Staubli VAL3: RobotPolish.pjx

--- RobotPolish.pjx ---
Parameters version=s7.3 stackSize=5000 millimeterUnit=true
Program file=DeleteTxt.pgx
Program file=Kill.pgx
Program file=Poll.pgx
Program file=_refreshDebugPa.pgx
Program file=alarm_action.pgx
Program file=checkIn.pgx
Program file=checkOut.pgx
Program file=check_PC.pgx
Program file=goHome.pgx
Program file=init.pgx
Program file=logandpopMsg.pgx
Program file=main.pgx
Program file=massage.pgx
Program file=page_debug.pgx
Program file=page_main.pgx
Program file=page_production.pgx
Program file=page_setHome.pgx
Program file=page_setSpdVal.pgx
Program file=page_txtSelect.pgx
Program file=prdMassage.pgx
Program file=prdStatusList.pgx
Program file=prd_action.pgx
Program file=production.pgx
Program file=readForce.pgx
Program file=resumeProduct.pgx
Program file=start.pgx
Program file=stop.pgx
Program file=userInterface.pgx
Data file=RobotPolish.dtx
Library alias=read path=Disk://readText/readText.pjx autoload=true password=
Library alias=io path=Disk://IO/IO.pjx autoload=true password=
Library alias=ati path=Disk://atiForceSen7/atiForceSen7.pjx autoload=true password=
Library alias=use path=Disk://userPage/userPage.pjx autoload=true password=
Library alias=date path=Disk://dateBase/dateBase.pjx autoload=true password=
Library alias=setFrm path=Disk://CircleCenter/CircleCenter.pjx autoload=true password=
Library alias=UI path=Disk://StaubliUI/StaubliUI.pjx autoload=true password=
Library alias=CalTool path=Disk://StaubliCalTool7/StaubliCalTool7.pjx autoload=true password=

--- RobotPolish.dtx ---
bool bBIO[32]
  [16] = true
  [18] = true
  [22] = true
bool bDebug_PC[6] = true
bool bExit = true
bool bForceError
bool bHome
bool bInterVal
bool bIsAlarm
bool bIsPower = true
bool bJntOrPtSpd
bool bOverRun
bool bPause
bool bRefreshMsg[6]
  [0] = true
  [1] = true
  [2] = true
  [3] = true
  [4] = true
  [5] = true
bool bSuspend = true
bool bTableAlm
bool bTxtLoad
bool bUpload
bool bZero
frame fFrame = {x=1612.970915, y=39.891118, z=-82.912831, rx=0.071185, ry=-0.543234, rz=-77.228709, fatherId=world[0]}
jointRx jCurrentJoint = {j1=8.22, j2=20.1, j3=107.19, j4=-141.77, j5=44.38, j6=150.9}
jointRx jHome = {j1=40.634813, j2=24.616005, j3=104.715218, j4=-108.663007, j5=68.526435, j6=132.709111}
jointRx jJHome = {j1=11.40774, j2=30.671658, j3=109.333141, j4=204.624689, j5=51.130912, j6=-196.428273}
mdesc mNomSpeed = {accel=36, vel=60, decel=36, rmax=2000, tmax=100, blend=cartesian, leave=5, reach=5}
num nATIPress
num nATiPressBuff
num nFunctionIndex = -1
num nInterfaceType = 9
num nJntList
public num nLimitAti[6]
  [0] = 500
  [1] = 500
  [2] = 500
  [3] = 100
  [4] = 100
  [5] = 100
num nMoveID
num nPage
num nPauseTime = 6
num nSelect
num nTabSpeed = 5
num nTimeBuff = 6728.108
num nTxtSelseted = 3
num nVirtualKey = -1
num nWorkModeStatus
num nWorkingMode = 4
pointRx p = {x=-96.25, y=181, rx=-8.631, ry=175.438, rz=-89.108, fatherId=fFrame[0]}
pointRx pCurrent = {x=-7.439422, y=-0.703489, z=141.92314, rx=-0.008216, ry=-179.493493, rz=-59.800957, shoulder=lefty, elbow=epositive, wrist=wpositive, fatherId=fFrame[0]}
string sButtons[2]
  [0] = "Yes"
  [1] = "No"
string sErrorMsg[8]
  [0] = "UPS报错，检查工厂供电"
  [1] = "转台故障报警"
  [2] = "工具报警"
  [3] = "ATI与机器人通讯异常"
  [4] = "打磨力超出上限"
  [5] = "急停状态激活中"
string sItems[8]
  [0] = "信号"
  [1] = "生产"
  [2] = "TCP"
  [3] = "Frame"
  [4] = "Home"
  [5] = "速度"
  [7] = "退出"
string sMassage
string sPrdStatus[10]
  [0] = "Txt文件:"
  [1] = "TEST.txt"
  [2] = "生产状态:无生产"
  [3] = "运动状态:Move"
  [4] = "总路径个数:     1"
  [5] = "当前路径  :     1"
  [6] = "写入点个数:   902"
  [7] = "读取点个数:     1"
  [8] = "当前MoveID:     0"
  [9] = "瞬时速度  :  5.4 "
string sStrFileName[6]
  [0] = "1233"
  [1] = "BUFF"
  [2] = "TEST.txt"
  [3] = "speed of TCP.txt"
string sTxtLists[12]
  [0] = "1233"
  [1] = "BUFF"
  [2] = "TEST"
  [3] = "TEST.txt"
  [4] = "speed of TCP.txt"
string sTxtSelected = "TEST.txt"
tool tTTool = {x=1.417, y=48.029, z=261.326, rx=-28.407, ry=-42.029, rz=-19.448, fatherId=flange[0], ioLink=valve1}
public tool tTool = {x=350.22, y=-0.767094, z=232.538993, rx=-89.841339, ry=89.729222, rz=89.842087, fatherId=flange[0], ioLink=valve1}
trsf trFrame = {x=1460.596362, y=35.712914, z=-199.189903, rx=-0.117127, ry=-0.30554, rz=-53.750077}

--- main.pgx ---
program main()
begin

  //初始化
  call DeleteTxt()
  call init()
  //创建同步任务,机器人实时读取ATI传感器数据
  //2015.06.23
  //taskCreateSync "readAtiForce",0.05,bOverRun,readForce()
  taskCreate "readAtiForce",100,readForce()


  //创建任务,实时扫描输入输出信号
  //当date:bPLC变量为true时,调用真实机器人联机调试程序;
  //当date:bPLC变量为false时,调用PC模拟程序;
  if date:bPLC
    taskCreate "Input",96,checkIn()
    taskCreate "Output",98,checkOut()
  else
    taskCreate "PC_IO",98,check_PC()
  endIf
  //创建任务,用户操作界面
  taskCreate "HMI",85,userInterface()



end

--- check_PC.pgx ---
program check_PC()
  local jointRx l_jCurrent
  local bool l_bRefresh
begin
  while !bExit

    //工厂断电报警
    if bDebug_PC[0]==false
      call logandpopMsg(sErrorMsg[0],bRefreshMsg[0])
      if read:bCycle
        call alarm_action()
      endIf
      if workingMode()==4
        disablePower()
      endIf
    else
      bRefreshMsg[0]=true
    endIf

    //check
    call Poll()
    //

    //转台故障信号
    //    if dioGet(io:doB_9_tableOn)==1
    //      if dioGet(io:doB_0_speed)==1 or dioGet(io:doB_1_speed)==1 or dioGet(io:doB_2_speed)==1 or dioGet(io:doB_3_speed)==1 or dioGet(io:doB_4_speed)==1 or dioGet(io:doB_5_speed)==1
    //        bTableAlm=!watch(dioGet(io:diB_2_tableOn)==1,2)
    //        if !bTableAlm
    //          bRefreshMsg[1]=true
    //        else
    //          call logandpopMsg(sErrorMsg[1],bRefreshMsg[1])
    //          if read:bCycle
    //            call alarm_action()
    //          endIf
    //        endIf
    //      else
    //        bTableAlm=false
    //      endIf
    //    else
    //      bTableAlm=false
    //    endIf
    //工具报警信号
    if bDebug_PC[2]==true
      call logandpopMsg(sErrorMsg[2],bRefreshMsg[2])
      if read:bCycle
        call alarm_action()
      endIf
    else
      bRefreshMsg[2]=true
    endIf
    //ATI通讯状态检测
    if bDebug_PC[3]==true
      call logandpopMsg(sErrorMsg[3],bRefreshMsg[3])
      if read:bCycle
        call alarm_action()
      endIf
    else
      bRefreshMsg[3]=true
    endIf
    //传感器力/扭矩上限检测
    //需要根据测试结果设置力及力矩上限
    if bDebug_PC[4]==true
      bForceError=true
      call logandpopMsg(sErrorMsg[4],bRefreshMsg[4])
      if read:bCycle
        call alarm_action()
      endIf
    else
      bForceError=false
      bRefreshMsg[4]=true
    endIf
    //急停处理
    if esStatus()==2
      call logandpopMsg(sErrorMsg[5],bRefreshMsg[5])
      call prd_action("急停处理")
    else
      bRefreshMsg[5]=true
    endIf
    //远程上电
    if workingMode(nWorkModeStatus)==4 and dioGet(io:diB_0_UPS)==0
      if dioGet(io:doB_10_systeAlm)==0
        enablePower()
        dioSet(io:doB_6_toolPower,1)
      else
        dioSet(io:doB_6_toolPower,0)
      endIf
    endIf
    //零位判断
    l_jCurrent=herej()
    if abs(l_jCurrent.j1-date:jHome.j1)<1 and abs(l_jCurrent.j2-date:jHome.j2)<1 and abs(l_jCurrent.j3-date:jHome.j3)<1 and abs(l_jCurrent.j4-date:jHome.j4)<2 and abs(l_jCurrent.j5-date:jHome.j5)<2 and abs(l_jCurrent.j6-date:jHome.j6)<2
      bHome=true
    else
      bHome=false
    endIf
    //系统报警信号判断
    if !bDebug_PC[0] or bTableAlm or bDebug_PC[2] or bDebug_PC[3] or bDebug_PC[4] or bDebug_PC[5]
      dioSet(io:doB_10_systeAlm,1)
    else
      dioSet(io:doB_10_systeAlm,0)
    endIf
    //报警处理
    if dioGet(io:doB_10_systeAlm)==1
      //
      call logandpopMsg("系统报警",l_bRefresh)
      if dioGet(io:doB_7_toolOn)==1
        dioSet(io:doB_7_toolOn,0)
      endIf
      if dioGet(io:doB_9_tableOn)==1
        dioSet(io:doB_9_tableOn,0)
      endIf
    else
      l_bRefresh=true
      call use:clear(0,12)
      delay(0)
    endIf
    delay(0)
  endWhile
end

--- DeleteTxt.pgx ---
program DeleteTxt()
  local num l_nNum
begin


  if libList("Disk://txt",sStrFileName)==false
    return
  endIf

  l_nNum=size(sStrFileName)
  if l_nNum<1
    return
  endIf

  for l_nNum=0 to size(sStrFileName)-1
    if find(sStrFileName[l_nNum],".txt")>0
      $delete("Disk://txt/"+sStrFileName[l_nNum])
    endIf


  endFor





  $fileClose(0)
  $fileClose(1)
  $fileClose(2)
  $fileClose(3)
  $fileClose(4)
  $fileClose(5)
  $fileClose(6)
  $fileClose(7)
  $fileClose(8)
  $fileClose(9)






end

--- page_debug.pgx ---
program page_debug()
  local string l_sItems
begin
  nPage=1
  cls()
  title("RobotPolish-调试页面")
  l_sItems="主轴上下电,主轴启停,转台启停,<-转台速度,->转台速度,编辑转台速度,置零ATI数据,返回上一级"
  call use:stringToArray(l_sItems,sItems)
  call use:setMenu(sItems,false,3)
  nInterfaceType=3
  gotoxy(0,11)
  put("转台当前速度："+toString("",nTabSpeed))
  if dioGet(io:doB_6_toolPower)==1
    gotoxy(15,3)
    put("[开]")
  else
    gotoxy(15,3)
    put("[关]")
  endIf
  if dioGet(io:doB_7_toolOn)==1
    gotoxy(13,4)
    put("[开]")
  else
    gotoxy(13,4)
    put("[关]")
  endIf
  if dioGet(io:doB_9_tableOn)==1
    gotoxy(13,5)
    put("[开]")
  else
    gotoxy(13,5)
    put("[关]")
  endIf
  if ati:bZero
    gotoxy(16,9)
    put("[开]")
  else
    gotoxy(16,9)
    put("[关]")
  endIf
  taskCreate "refDedugpage",50,_refreshDebugPa()
end

--- page_setHome.pgx ---
program page_setHome()
  local num l_nNum[6]
  local string l_sString[6]
  local num i
  local string l_sStr[6]
  local num l_nKey
  local joint l_CurrentJ
  local bool bHere
  local bool l_bExit
begin
  bHere=false
  l_bExit=false
  title("RobotPolish-Home示教页面")
  cls()
  call use:stringToArray("记录当前位置,移动至记录点,,,,保存并上传数据,,返回上一级",sItems)
  call use:setMenu(sItems,true,3)
  l_sString[0]="J1"
  l_sString[1]="J2"
  l_sString[2]="J3"
  l_sString[3]="J4"
  l_sString[4]="J5"
  l_sString[5]="J6"
  l_nNum[0]=jHome.j1
  l_nNum[1]=jHome.j2
  l_nNum[2]=jHome.j3
  l_nNum[3]=jHome.j4
  l_nNum[4]=jHome.j5
  l_nNum[5]=jHome.j6
  //Create the LIST
  call use:setSizeList(20,3,15,6)
  call use:listcreate("Home关节位置")
  //Insert Items
  for i=0 to 5
    call use:strlength(l_sString[i],3)
    l_sString[i]=l_sString[i]+":"+toString("8.3",l_nNum[i])
    call use:listadd(l_sString[i])
  endFor
  call use:listupdate(0)
  call use:listcursor(nJntList,true)
  while !l_bExit
    l_nKey=getKey()
    switch l_nKey
      case 261
        if nJntList>0
          call use:listcursor(nJntList,false)
          nJntList=nJntList-1
          call use:listcursor(nJntList,true)
        elseIf nJntList==0
          call use:listcursor(nJntList,false)
          nJntList=5
          call use:listcursor(nJntList,true)
        endIf
      break
      case 266
        if nJntList<5
          call use:listcursor(nJntList,false)
          nJntList=nJntList+1
          call use:listcursor(nJntList,true)
        elseIf nJntList==5
          call use:listcursor(nJntList,false)
          nJntList=0
          call use:listcursor(nJntList,true)
        endIf
      break
      case 270
        call use:changeValue(l_nNum[nJntList],-270,270,26,4+nJntList,l_sStr)
        jHome.j1=l_nNum[0]
        jHome.j2=l_nNum[1]
        jHome.j3=l_nNum[2]
        jHome.j4=l_nNum[3]
        jHome.j5=l_nNum[4]
        jHome.j6=l_nNum[5]
        //Create the LIST
        call use:setSizeList(20,3,15,6)
        call use:listcreate("Home关节位置")
        //Insert Items
        for i=0 to 5
          call use:strlength(l_sString[i],3)
          l_sString[i]=l_sString[i]+":"+toString("8.3",l_nNum[i])
          call use:listadd(l_sString[i])
        endFor
        call use:listupdate(0)
        call use:listcursor(nJntList,true)
      break
      case 271
        call use:questionDialog("确定记录当前位置?",sButtons,l_nKey)
        if (l_nKey==0 or l_nKey==1) and herej()!={0,0,0,0,0,0}
          jHome=herej()

          l_nNum[0]=jHome.j1
          l_nNum[1]=jHome.j2
          l_nNum[2]=jHome.j3
          l_nNum[3]=jHome.j4
          l_nNum[4]=jHome.j5
          l_nNum[5]=jHome.j6
          cls()
          call use:stringToArray("记录当前位置,移动至记录点,,,,保存并上传数据,,返回上一级",sItems)
          call use:setMenu(sItems,true,3)
          //Create the LIST
          call use:setSizeList(20,3,15,6)
          call use:listcreate("Home关节位置")
          //Insert Items
          for i=0 to 5
            call use:strlength(l_sString[i],3)
            l_sString[i]=l_sString[i]+":"+toString("8.3",l_nNum[i])
            call use:listadd(l_sString[i])
          endFor
          call use:listupdate(0)
          call use:listcursor(nJntList,true)
          call massage("记录完成!")
          bHere=true
        else
          if herej()=={0,0,0,0,0,0}
            popUpMsg("安全点不能全为零")
          endIf
          cls()
          call use:stringToArray("记录当前位置,移动至记录点,,,,保存并上传数据,,返回上一级",sItems)
          call use:setMenu(sItems,true,3)
          //Create the LIST
          call use:setSizeList(20,3,15,6)
          call use:listcreate("Home关节位置")
          //Insert Items
          for i=0 to 5
            call use:strlength(l_sString[i],3)
            l_sString[i]=l_sString[i]+":"+toString("8.3",l_nNum[i])
            call use:listadd(l_sString[i])
          endFor
          call use:listupdate(0)
          call use:listcursor(nJntList,true)
        endIf
      break
      case 272
        l_CurrentJ=herej()
        if abs(l_CurrentJ.j1-jHome.j1)>1 or abs(l_CurrentJ.j2-jHome.j2)>1 or abs(l_CurrentJ.j3-jHome.j3)>1 or abs(l_CurrentJ.j4-jHome.j4)>1 or abs(l_CurrentJ.j5-jHome.j5)>1 or abs(l_CurrentJ.j6-jHome.j6)>1
          popUpMsg("按Move-Hold键回零位")
          resetMotion()
          movej(jHome,flange,mNomSpeed)
          waitEndMove()
          call massage("到达Home位置!")
        else
          popUpMsg("手臂已在当前位置")
        endIf
      break
      case 276
        date:jHome=jHome
        libSave()
        date:libSave()
        bUpload=true
        call massage("数据上传完成!")
        bHere=false
      break
      case 278
        if bHere==true
          call use:questionDialog("为保存修改数据,确定返回?",sButtons,l_nKey)
          if l_nKey==0 or l_nKey==1
            l_bExit=true
          else
            cls()
            call use:stringToArray("记录当前位置,移动至记录点,,,,保存并上传数据,,返回上一级",sItems)
            call use:setMenu(sItems,true,3)
            //Create the LIST
            call use:setSizeList(20,3,15,6)
            call use:listcreate("Home关节位置")
            //Insert Items
            for i=0 to 5
              call use:strlength(l_sString[i],3)
              l_sString[i]=l_sString[i]+":"+toString("8.3",l_nNum[i])
              call use:listadd(l_sString[i])
            endFor
            call use:listupdate(0)
            call use:listcursor(nJntList,true)
          endIf
        else
          l_bExit=true
        endIf
      break
    endSwitch
    delay(0)
  endWhile
  call page_main()
end

--- page_setSpdVal.pgx ---
program page_setSpdVal()
  local num i
  local num l_nKey
  local string l_sString[7]
  local num l_nNum[7]
  local string l_sStr
  local num nMspdList
begin
  title("RobotPolish-设定速度参数默认值")
  cls()
  l_sString[0]="加速度(%)"
  l_sString[1]="速度(%)"
  l_sString[2]="减速度(%)"
  l_sString[3]="Tvel(mm/s)"
  l_sString[4]="转速(deg/s)"
  l_sString[5]="Leave(mm)"
  l_sString[6]="Reach(mm)"
  l_nNum[0]=date:mGrindingSpd.accel
  l_nNum[1]=date:mGrindingSpd.vel
  l_nNum[2]=date:mGrindingSpd.decel
  l_nNum[3]=date:mGrindingSpd.tvel
  l_nNum[4]=date:mGrindingSpd.rvel
  l_nNum[5]=date:mGrindingSpd.leave
  l_nNum[6]=date:mGrindingSpd.reach
  //Create the LIST
  call use:setSizeList(10,3,20,7)
  call use:listcreate("Set_mPointSpeed")
  //Insert Items
  for i=0 to 6
    call use:strlength(l_sString[i],11)
    l_sString[i]=l_sString[i]+":"+toString("8.3",l_nNum[i])
    call use:listadd(l_sString[i])
  endFor
  call use:typeMenu(6,"上传")
  call use:typeMenu(8,"返回")
  call use:listupdate(0)
  call use:listcursor(nMspdList,true)
  do
    l_nKey=getKey()
    switch l_nKey
      case 261
        if nMspdList>0
          call use:listcursor(nMspdList,false)
          nMspdList=nMspdList-1
          call use:listcursor(nMspdList,true)
        elseIf nMspdList==0
          call use:listcursor(nMspdList,false)
          nMspdList=6
          call use:listcursor(nMspdList,true)
        endIf
      break
      case 266
        if nMspdList<6
          call use:listcursor(nMspdList,false)
          nMspdList=nMspdList+1
          call use:listcursor(nMspdList,true)
        elseIf nMspdList==6
          call use:listcursor(nMspdList,false)
          nMspdList=0
          call use:listcursor(nMspdList,true)
        endIf
      break
      case 270
        call use:changeValue(l_nNum[nMspdList],0,99999,23,4+nMspdList,l_sStr)
        date:mGrindingSpd.accel=l_nNum[0]
        date:mGrindingSpd.vel=l_nNum[1]
        date:mGrindingSpd.decel=l_nNum[2]
        date:mGrindingSpd.tvel=l_nNum[3]
        date:mGrindingSpd.rvel=l_nNum[4]
        date:mGrindingSpd.leave=l_nNum[5]
        date:mGrindingSpd.reach=l_nNum[6]
        //Create the LIST
        call use:setSizeList(10,3,20,7)
        call use:listcreate("Set_mPointSpeed")
        //Insert Items
        for i=0 to 6
          call use:strlength(l_sString[i],11)
          l_sString[i]=l_sString[i]+":"+toString("8.3",l_nNum[i])
          call use:listadd(l_sString[i])
        endFor
        call use:listupdate(0)
        call use:listcursor(nMspdList,true)
        date:libSave()
      break
      case 276
        //Joint类型速度参数定义
        for l_nNum=0 to 99
          read:mSpdOfJnt[l_nNum].accel=16
          read:mSpdOfJnt[l_nNum].vel=40
          read:mSpdOfJnt[l_nNum].decel=16
          read:mSpdOfJnt[l_nNum].tvel=200
          read:mSpdOfJnt[l_nNum].rvel=1000
          read:mSpdOfJnt[l_nNum].blend=Cartesian
          read:mSpdOfJnt[l_nNum].leave=2
          read:mSpdOfJnt[l_nNum].reach=2
        endFor
        for i=0 to size(read:mSpdOfPt)-1
          read:mSpdOfPt[i].vel=date:mGrindingSpd.vel
          read:mSpdOfPt[i].accel=date:mGrindingSpd.accel
          read:mSpdOfPt[i].decel=date:mGrindingSpd.decel
          read:mSpdOfPt[i].leave=date:mGrindingSpd.leave
          read:mSpdOfPt[i].reach=date:mGrindingSpd.reach
          read:mSpdOfPt[i].tvel=date:mGrindingSpd.tvel
          read:mSpdOfPt[i].rvel=date:mGrindingSpd.rvel
          read:mSpdOfPt[i].blend=date:mGrindingSpd.blend
        endFor
        //read:libSave()
        call massage("数据上传完成!")
      break
    endSwitch
    delay(0)
  until l_nKey==278 or l_nKey==255
  call page_main()
end

--- page_txtSelect.pgx ---
program page_txtSelect()
begin
  cls()
  nPage=3
  title("RobotPolish-生产页面-.Txt选择")
  libList("Disk://txt",sTxtLists)
  call use:setSizeList(2,0,36,10)
  call use:listcreate("Txt Lists")
  call use:listadd(sTxtLists)
  if size(sTxtLists)<=10
    call use:listupdate(0)
  else
    if nTxtSelseted>9
      call use:listupdate(nTxtSelseted-9)
    else
      call use:listupdate(0)
    endIf
  endIf
  call massage("提示：上下键选择Txt文件")
  call use:typeMenu(8,"OK")
end

--- production.pgx ---
program production()
begin
  if taskStatus("txtLoad")!=-1
    taskKill("txtLoad")
    wait(taskStatus("txtLoad")==-1)
  endIf
  if taskStatus("motion")!=-1
    taskKill("motion")
    wait(taskStatus("motion")==-1)
  endIf
  //2015.06.23
  //taskCreateSync "txtLoad",0.004,bTxtLoad,read:fileRead(sTxtSelected)
  taskCreate "txtLoad",100,read:fileRead(sTxtSelected)
  taskCreate "motion",98,read:trajGrind()
  if taskStatus("prdMassage")==-1
    taskCreate "prdMassage",80,prdMassage()
  endIf
end
